(* IEC 61131-3 sources: Py_iec/tests/fixtures/st/invalid, 1 file *)

(* ---- missing_target.st ---- *)
FUNCTION_BLOCK Counter
VAR
    count : INT := 0;
END_VAR
missing := count + 1;
END_FUNCTION_BLOCK
